# EPICS substitutions: streamApp/pluginDb/pluginColorConvert.substitutions
#
# pluginColorConvert.substitutions
#

file NDPluginBase.template
{
	{
	P=$(CAM):,
	R=CC$(N):,
	PORT=CC$(N),
	ADDR=0,
	TIMEOUT=1,
	NDARRAY_PORT=$(PLUGIN_SRC),
	NDARRAY_ADDR=0,
	}
}

file NDColorConvert.template
{
	{
	P=$(CAM):,
	R=CC$(N):,
	PORT=CC$(N),
	ADDR=0,
	TIMEOUT=1
	}
}
